FUNCTION_BLOCK Q_SetAudioVolume (* Command SetAudioVolume. *)
  (* Standard: ISO 11783-6; Description: This command can be used to control the audio on the VT (volume) ( Part 6 - F.12 ) Return values iso_s16 - E_NO_ERR - OK - E_OVERFLOW - Buffer overflow - E_NOACT - Command not possible in current state - E_NOT_AVAILABLE - VT has got no adjustable volume output - E_NO_INSTANCE - No VT client available *)
  (* Version 1.0, 2022-07-08, franz *)
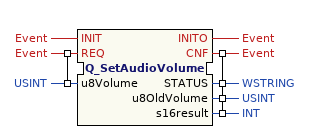
  EVENT_INPUT
    INIT; (* Service Initialization *)
    REQ WITH u8Volume; (* Service Request *)
  END_EVENT
  EVENT_OUTPUT
    INITO; (* Initialization Confirm *)
    CNF WITH STATUS, s16result, u8OldVolume; (* Confirmation of Requested Service *)
  END_EVENT
  VAR_INPUT
    u8Volume : USINT; (* Volume 0 - 100 (%) *)
  END_VAR
  VAR_OUTPUT
    STATUS : WSTRING; (* Service Status *)
    u8OldVolume : USINT; (* Old volume 0 - 100 (%) *)
    s16result : INT; (* retval see description *)
  END_VAR
END_FUNCTION_BLOCK
